PROGRAM MAIN
VAR
iVolt 		AT%I* : UINT;
iTempSens1 	AT%Q* : UINT;
iTempSens2 	AT%Q* : UINT;
fbTempModel : Temp_Model0;
END_VAR


fbTempModel(ssMethodType:= , iVolt_U:= iVolt , iTemp1_Y=> iTempSens1 , iTemp2_Y=> iTempSens2 );
fbTempModel.ssMethodType := 1;

END_PROGRAM

(* stored: Version 1.1.0.1, ProductVersion 3.1.4024.13
   POU MAIN: Id {73325dd8-e90f-4efc-b2df-427ecaf831ca}, SpecialFunc None *)
